KUKA KRL program: FrameDataAut3.src, FrameDataAut3.dat

--- FrameDataAut3.src ---
&ACCESS RVO2
&REL 3
DEFFCT ST_Dim3 FrameDataAut3(eElement:IN,iElement:IN)
   ;FOLD DECL
      DECL Data_FrameAut3 eElement
      DECL INT iElement
      DECL ST_Dim3 stData
   ;ENDFOLD (DECL)

   SWITCH eElement
      CASE #Plate
         stData = GetPlatePlace(iElement)
      CASE #Screw
         stData = GetScrewPlace(iElement)
      CASE #Pocket
         stData = GetPocketPlace(iElement)
      CASE #PocketDim
         stData = GetPocketDim(iElement)
      DEFAULT
         HALT
   ENDSWITCH

   RETURN stData

ENDFCT

DEFFCT ST_Dim3 GetPlatePlace(iPlate:IN)
   ;FOLD DECL
      DECL INT iPlate
      DECL ST_Dim3 stPlate
      DECL E_ProfileType eProfileType
   ;ENDFOLD (DECL)

   ;ProcessData
   eProfileType = gstProcessData.eProfileType

   ;stPlate
   SWITCH eProfileType
      CASE #Frame75
         stPlate = stPlateFrame75[iPlate]
      CASE #Frame90
         stPlate = stPlateFrame90[iPlate]
      DEFAULT
         HALT
   ENDSWITCH

   ;Return plate place
   RETURN stPlate

ENDFCT

DEFFCT ST_Dim3 GetScrewPlace(iScrew:IN)
   ;FOLD DECL
      DECL INT iScrew,iPlate,iScrewDist
      DECL ST_Dim3 stPlate,stScrew
      DECL REAL rScrewOffsetDist
   ;ENDFOLD (DECL)

   ;iPlate,rScrewOffsetDist
   SWITCH iScrew
      CASE 1,2
         iPlate = 1
         iScrewDist = iScrew
         rScrewOffsetDist = rAuxPlateScrewDist[iScrewDist]
      CASE 3,4,5
         iPlate = 2
         iScrewDist = iScrew - 2
         rScrewOffsetDist = rMainPlateScrewDist[iScrewDist]
      CASE 6,7
         iPlate = 3
         iScrewDist = iScrew - 5
         rScrewOffsetDist = rAuxPlateScrewDist[iScrewDist]
      DEFAULT
         HALT
   ENDSWITCH

   ;stPlate
   stPlate = GetPlatePlace(iPlate)

   ;stScrew
   stScrew.rX = stPlate.rX + rScrewOffsetDist
   stScrew.rY = stPlate.rY

   ;Return screw data
   RETURN stScrew

ENDFCT

DEFFCT ST_Dim3 GetPocketPlace(iPocket:IN)
   ;FOLD DECL
      DECL INT iPocket,iPlate
      DECL ST_Dim3 stPocket,stPlate,stPocketOffset
   ;ENDFOLD (DECL)

   ;iPlate
   SWITCH iPocket
      CASE 1,2,3
         iPlate = iPocket
      DEFAULT
         HALT
   ENDSWITCH

   ;stPlate
   stPlate = GetPlatePlace(iPlate)

   ;stPocketOffset
   SWITCH iPocket
      CASE 1,3
         stPocketOffset = {rX 0.0,rY 0.0}
      CASE 2
         stPocketOffset.rX = stMainPocketOffset.rX
         stPocketOffset.rY = stMainPocketOffset.rY
      DEFAULT
         HALT
   ENDSWITCH

   ;stPocketOut
   stPocket.rX = stPlate.rX + stPocketOffset.rX
   stPocket.rY = stPlate.rY + stPocketOffset.rY

   ;Return pocket place
   RETURN stPocket

ENDFCT

DEFFCT ST_Dim3 GetPocketDim(iPocket:IN)
   ;FOLD DECL
      DECL INT iPocket
      DECL ST_Dim3 stPocketDim
   ;ENDFOLD (DECL)

   ;stPocketDim
   SWITCH iPocket
      CASE 1,3
         stPocketDim = stAuxPocketDim
      CASE 2
         stPocketDim = stMainPocketDim
      DEFAULT
         HALT
   ENDSWITCH

   ;Return pocket dimensions
   RETURN stPocketDim

ENDFCT

--- FrameDataAut3.dat ---
&ACCESS RVO2
&REL 3
DEFDAT FrameDataAut3 PUBLIC

   GLOBAL ENUM Data_FrameAut3 Plate,Screw,Pocket,PocketDim

   ;Okucie jako plate? AuxPlate i MainPlate?

   ;Plates placement Frame75 - Tablice czy main, aux?
   DECL CONST ST_Dim3 stPlateFrame75[3]
   stPlateFrame75[1] = {rX  270.0,rY 54.5} ;Bottom aux plate
   stPlateFrame75[2] = {rX 1017.0,rY 54.5} ;Main plate
   stPlateFrame75[3] = {rX 1760.0,rY 54.5} ;Upper aux plate

   ;Plates placement Frame90
   DECL CONST ST_Dim3 stPlateFrame90[3]
   stPlateFrame90[1] = {rX  275.0,rY 67.0} ;Bottom aux plate
   stPlateFrame90[2] = {rX 1022.0,rY 67.0} ;Main plate
   stPlateFrame90[3] = {rX 1765.0,rY 67.0} ;Upper aux plate

   ;AuxPlate data
   DECL CONST ST_Dim3 stAuxPocketDim = {rX 73.0,rY 18.0}
   DECL CONST REAL rAuxPlateScrewDist[2]
   rAuxPlateScrewDist[1] = -48.0
   rAuxPlateScrewDist[2] = +48.0

   ;MainPlate data
   DECL CONST ST_Dim3 stMainPocketDim = {rX 73.0,rY 18.0}
   DECL CONST ST_Dim3 stMainPocketOffset = {rX -53.0,rY 0.0}
   DECL CONST REAL rMainPlateScrewDist[3]
   rMainPlateScrewDist[1] = -96.0
   rMainPlateScrewDist[2] =  -5.0
   rMainPlateScrewDist[3] =  96.5

ENDDAT
